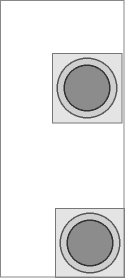
VISUALIZATION Visualization  // 125x278
    PushSwitchLed (52,53 70x70), variable: SyncProgram.bStartButton, behaviour: TAP, style: Switch-PushSwitchLed-Gray
    PushSwitchLed (55,208 70x70), variable: SyncProgram.bStopButton, behaviour: TAP, style: Switch-PushSwitchLed-Gray
END_VISUALIZATION

(* stored: Version 1.1.0.1, ProductVersion 3.1.4024.12
   Visu Visualization: Id {8b122034-5517-456f-8d92-653081f8c1ef} *)
